PROGRAM MAIN
VAR
END_VAR

END_PROGRAM

(* stored: Version 1.1.0.1
   POU MAIN: Id {52eff828-3ee9-4321-a8ed-fc53bb299b1f} *)
